FUNCTION_BLOCK FB_Observable_DINT EXTENDS FB_AbstractObservable
VAR
    _nVal:              DINT;
    _nOldVal:           DINT;
END_VAR

METHOD FB_init : BOOL
VAR_INPUT
    bInitRetains:       BOOL; // if TRUE, the retain variables are initialized (warm start / cold start)
    bInCopyCode:        BOOL;  // if TRUE, the instance afterwards gets moved into the copy code (online change)
END_VAR
THIS^._nTypeClass := __SYSTEM.TYPE_CLASS.TYPE_DINT;
END_METHOD

PROPERTY nDataSize : UDINT
GET
nDataSize := SIZEOF(DINT);
END_GET
END_PROPERTY

PROPERTY nValue32 : DINT
GET
nValue32 := THIS^._nVal;
END_GET
SET
THIS^._nOldVal := THIS^._nVal;
THIS^._nVal := nValue32;

THIS^.NotifyWithConditions();
END_SET
END_PROPERTY

PROPERTY PROTECTED pData : POINTER TO BYTE
GET
pData := ADR(THIS^._nVal);
END_GET
END_PROPERTY

METHOD  ValueChanged : BOOL
VAR_INPUT
END_VAR
ValueChanged := THIS^._nOldVal <> THIS^._nVal;
END_METHOD

END_FUNCTION_BLOCK

(* stored: Version 1.1.0.1, ProductVersion 3.1.4024.12
   POU FB_Observable_DINT: Id {6de3a4c4-474b-46c8-abeb-2912757def04}, SpecialFunc None
   Method FB_init: Id {6962c5dd-d23f-0cfe-06d1-b81f49c6f4dc}
   Property nDataSize: Id {4c034ca1-003d-47b0-8cb3-b0f6f52bcea9}
   Get Get: Id {3d907f8e-1f44-4da0-afe1-b39929fb8aef}
   Property nValue32: Id {8c6e5650-be92-461f-8538-94a03dc98106}
   Get Get: Id {8fd5783a-ed1c-4ca8-980a-76c10d0027c7}
   Set Set: Id {7690aef0-1b32-4f34-b842-7c699fcf50f7}
   Property pData: Id {9b5bca01-fad3-4c25-9c57-3ea842b8ebf4}
   Get Get: Id {ff883c77-6cfc-480c-8763-70e9f38ec28b}
   Method ValueChanged: Id {828a2292-a65c-099b-1ba9-cf732316f206} *)
